Universal Robots PolyScope program: MATEO.urp

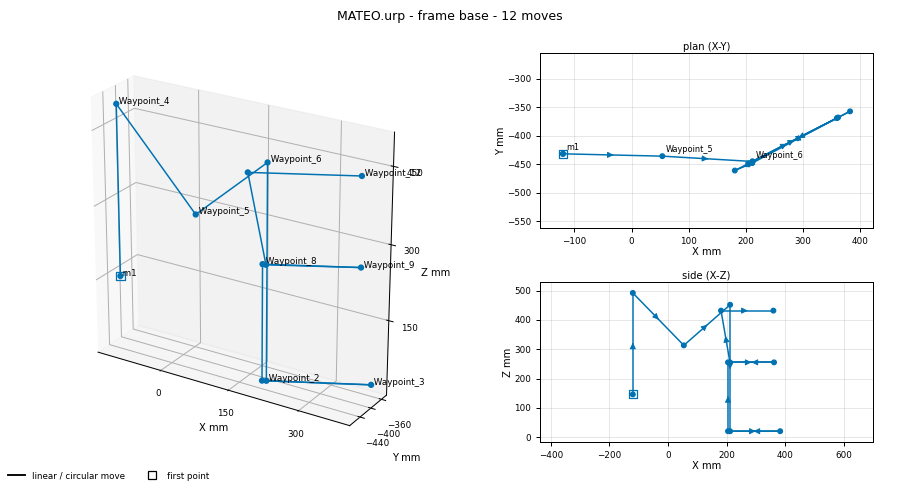
[picture p0: tool path of MATEO.urp in frame base, 12 of 12 moves have a stored position in this frame; points joined in program order, loops and branches not executed]
Program name (installation=default directory=/ursim/programs createdIn=3.15.8.106339 lastSavedIn=3.15.8.106339 robotSerialNumber=2018359999)
Calibrated DH parameters: a=[0, -0.425, -0.39225, 0, 0, 0]; d=[0.089159, 0, 0, 0.10915, 0.09465, 0.0823]; alpha=[1.570796, 0, 0, 1.570796, -1.570796, 0]; deltaTheta=[0, 0, 0, 0, 0, 0]
Robot Program (runOnlyOnce=false)
  Popup Message (haltProgram=false message=Se va a simular la M inputType=Text)
  MoveL speed 250 mm/s, acceleration 1200 mm/s^2 (useActiveTCP=true) feature=Base
    Waypoint m1: TCP in base x=-120.113 y=-431.763 z=146.073 mm, rx=-0.0012 ry=3.1163 rz=0.0389 rad; joints [-91.713, -98.956, -126.223, -46.295, 91.393, -1.776] deg
    Waypoint Waypoint_4: TCP in base x=-120.113 y=-431.763 z=492.071 mm, rx=-0.0012 ry=3.1163 rz=0.0389 rad; joints [-91.713, -84.032, -86.444, -100.996, 91.393, -1.776] deg
    Waypoint Waypoint_5: TCP in base x=53.835 y=-435.868 z=313.273 mm, rx=-0.0012 ry=3.1163 rz=0.0389 rad; joints [-68.927, -84.281, -112.793, -73.744, 91.854, 21.015] deg
    Waypoint Waypoint_6: TCP in base x=211.664 y=-445.145 z=451.776 mm, rx=-0.0012 ry=3.1163 rz=0.0389 rad; joints [-52.12, -89.366, -87.667, -93.214, 92.012, 37.831] deg
    Waypoint Waypoint_2: TCP in base x=211.664 y=-445.145 z=20.542 mm, rx=-0.0012 ry=3.1163 rz=0.0389 rad; joints [-52.12, -120.397, -123.599, -26.252, 92.012, 37.831] deg
    Popup Message (haltProgram=false message=Se va a simular la letra E inputType=Text)
  MoveL speed 250 mm/s, acceleration 1200 mm/s^2 (useActiveTCP=true) feature=Base
    Waypoint Waypoint_3: TCP in base x=382.44 y=-357.401 z=20.541 mm, rx=-0.0012 ry=3.1163 rz=0.0389 rad; joints [-31.342, -122.744, -118.731, -28.043, 91.969, 58.621] deg
    Waypoint Waypoint_7: TCP in base x=204.548 y=-448.801 z=20.541 mm, rx=-0.0012 ry=3.1163 rz=0.0389 rad; joints [-53.056, -120.415, -123.54, -26.325, 92.008, 36.894] deg
    Waypoint Waypoint_8: TCP in base x=204.548 y=-448.801 z=255.34 mm, rx=-0.0012 ry=3.1163 rz=0.0389 rad; joints [-53.056, -94.876, -111.551, -63.854, 92.008, 36.894] deg
    Waypoint Waypoint_9: TCP in base x=361.448 y=-368.186 z=255.34 mm, rx=-0.0012 ry=3.1163 rz=0.0389 rad; joints [-33.64, -97.811, -108.407, -63.378, 91.986, 56.322] deg
    Waypoint Waypoint_10: TCP in base x=211.227 y=-447.981 z=255.34 mm, rx=-0.0012 ry=3.1163 rz=0.0389 rad; joints [-52.367, -95.148, -111.256, -63.852, 92.011, 37.584] deg
    Waypoint Waypoint_11: TCP in base x=180.71 y=-461.049 z=431.74 mm, rx=-0.0012 ry=3.1163 rz=0.0389 rad; joints [-56.202, -89.639, -90.291, -90.461, 91.989, 33.746] deg
    Waypoint Waypoint_12: TCP in base x=359.313 y=-369.283 z=431.74 mm, rx=-0.0012 ry=3.1163 rz=0.0389 rad; joints [-33.878, -92.251, -87.821, -89.533, 91.988, 56.084] deg
